(* PLC project Unnamed, Unknown Unnamed 1 *)
(* stored: creationDateTime 2026-03-14T10:04:09, modificationDateTime 2026-03-14T10:04:09 *)

PROGRAM main
  VAR
    Discharge AT %IX100.0 : BOOL := 1;
    I_Fill AT %IX100.1 : BOOL;
    Discharge_valve AT %QX100.0 : BOOL;
    Discharging AT %QX100.1 : BOOL;
    Fill_valve AT %QX100.2 : BOOL;
    Filling AT %QX100.3 : BOOL;
    Timer AT %QW100 : INT;
  END_VAR
  VAR
    TOF0 : TOF;
    TOF1 : TOF;
    fill_time_to_count : TIME;
    discharge_time_to_count : TIME;
    only_dis : BOOL;
    only_fill : BOOL;
  END_VAR

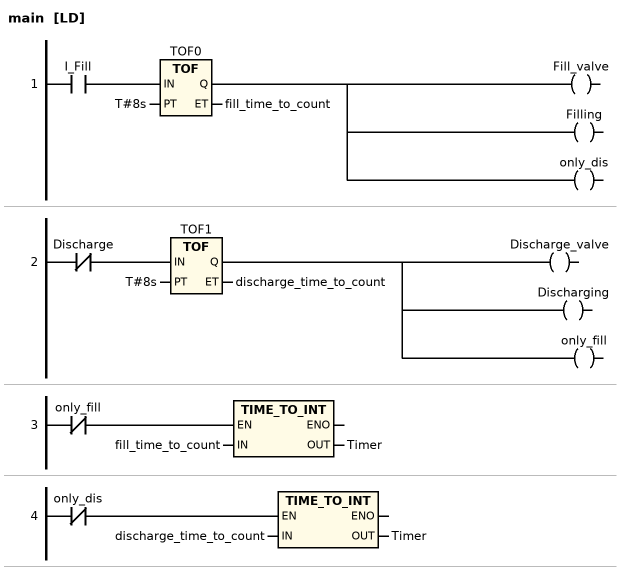
(* LD diagram, written out as Structured Text *)
TOF0(IN := I_Fill, PT := T#8s);
Fill_valve := TOF0.Q;
Filling := TOF0.Q;
only_dis := TOF0.Q;
TOF1(IN := NOT Discharge, PT := T#8s);
Discharge_valve := TOF1.Q;
Discharging := TOF1.Q;
only_fill := TOF1.Q;
fill_time_to_count := TOF0.ET;
discharge_time_to_count := TOF1.ET;
IF NOT only_fill THEN Timer := TIME_TO_INT(fill_time_to_count); END_IF;
IF NOT only_dis THEN Timer := TIME_TO_INT(discharge_time_to_count); END_IF;
END_PROGRAM

CONFIGURATION Config0
  RESOURCE Res0 ON PLC
    TASK task0(INTERVAL := T#20ms, PRIORITY := 1);
    PROGRAM instance0 WITH task0 : main;
  END_RESOURCE
END_CONFIGURATION
